TEXTLIST TL_E_MESSAGETYPE
  0 = 'eMessageEmpty'
  1 = 'eMessageError'
  2 = 'eMessageWarning'
  3 = 'eMessageInfo'
  4 = 'eMessageVerbose'
   = ''
END_TEXTLIST

(* stored: Version 1.1.0.1, ProductVersion 3.1.4026.13
   TextList TL_E_MESSAGETYPE: Id {f0419335-f227-4c5e-ab76-e1f19fdc6038} *)
